TYPE STATION_DONE :
STRUCT
		POSITION_DONE				: ARRAY[0..35] OF BOOL;
END_STRUCT
END_TYPE

(* stored: Version 1.1.0.1, ProductVersion 3.1.4024.11
   DUT STATION_DONE: Id {edbac3c1-fe99-4562-97aa-344905bb2b74} *)
